// TIA Portal V21 export
TYPE "LBC_typeMotorStarterCommandStates"
TITLE = LBC_typeMotorStarterCommands
// Module related manual commands from HMI
   STRUCT
      reset : Bool;   // Manual reset command from HMI,TRUE: Reset the motor starter. Output `resetStarter` is TRUE at least for the time configured at parameter `resetTime`
      commandForward : Bool;   // Manual forward command from HMI, Rising edge: Start the motor forward
      commandBackward : Bool;   // Manual backward command from HMI, Rising edge: Start the motor backward
   END_STRUCT;
END_TYPE
